(* IEC 61131-3 sources: IceManRemastered/Device/application/Motors, 3 files *)

(* ---- MotorOverride.st ---- *)
TYPE MotorOverride :
STRUCT
	Override: BOOL;
	Forward: BOOL;
	Reverse: BOOL;
	Brake: BOOL;
END_STRUCT
END_TYPE

(* ---- Motors.gvl.st ---- *)
{attribute 'qualified_only'}
VAR_GLOBAL
	AgitatorMotor: AgitatorMotor;
	BagFeedMotor: BagFeedMotor;
	BagFeedMotor_: BagFeedMotor_;
	BlowerMotor: BlowerMotor;
	HeatSealMotor: HeatSealMotor;
	IceFeedMotor: IceFeedMotor;
	KickerMotor: KickerMotor;
END_VAR

(* ---- EdgeTracker.st ---- *)
FUNCTION_BLOCK EdgeTracker
VAR_INPUT
	Trigger: 			BOOL;				//
	Triggers: 			UINT;				//
	Count: 				UDINT;				//
END_VAR
VAR_OUTPUT
	Edges: 				ARRAY[0..100] OF UDINT;
END_VAR
VAR
END_VAR

// --- BEGIN IMPLEMENTATION ---

IF Trigger = TRUE THEN
	Edges[Triggers]:=Count;
END_IF
